{attribute 'reflection'}
FUNCTION_BLOCK ABSTRACT Objective
VAR_INPUT

	Mediator					: REFERENCE TO Mediator;	

END_VAR
VAR

    internalRegisteredMoverCount 	: USINT;
   
    internalRegisteredMovers 		: ARRAY[1..Param.NUM_MOVERS] OF POINTER TO Mover;

	{attribute 'hide'}
    ErrorMover 					: ErrorMover;
	
    {attribute 'instance-path'}
    {attribute 'noinit'}
    InstancePath 				: STRING; // Unique variable path of the instance	
END_VAR
VAR_OUTPUT
END_VAR

PROPERTY CurrentMover : Reference to Mover
GET

// If no real mover can be returned as Current, return an imposter instead to output error messages
IF __ISVALIDREF( CurrentMover ) = FALSE THEN
	ErrorMover.SourceInstancePath	:= THIS^.InstancePath;
	CurrentMover					REF= ErrorMover;
END_IF
END_GET
END_PROPERTY

{attribute 'monitoring' := 'call'}
PROPERTY RegisteredMoverCount : USINT
GET
VAR
    i : INT;
END_VAR
RegisteredMoverCount := 0;

FOR i := 1 to Param.NUM_MOVERS DO

    IF internalRegisteredMovers[i] <> 0 THEN
        RegisteredMoverCount := RegisteredMoverCount + 1;
    END_IF

END_FOR
END_GET
END_PROPERTY

PROPERTY RegisteredMovers : ARRAY[0..Param.NUM_MOVERS - 1] OF POINTER TO Mover
GET
RegisteredMovers := internalRegisteredMovers;
END_GET
END_PROPERTY

METHOD RegisterMover : BOOL
VAR_INPUT
    NewMover : REFERENCE TO Mover;
END_VAR

VAR
    i              : ULINT;
    duplicateFound : BOOL;
    emptyIDX       : ulint;
END_VAR
(*
	Add a mover to a list of movers tracked by the objective.
	Movers can't be added multiple times, so check for duplicates
	Movers can't overwrite others in the list, so check that the array element is clear
*)

IF __ISVALIDREF(NewMover) THEN // validate reference

    duplicateFound            := FALSE; // default to false, counterexample below
    internalRegisteredMoverCount := 0;     // reset to zero, incremented below

    FOR i := 1 TO SIZEOF(internalRegisteredMovers) / SIZEOF(internalRegisteredMovers[i]) DO
        IF internalRegisteredMovers[i] <> 0 THEN
            IF ADR(NewMover) = internalRegisteredMovers[i] THEN
                duplicateFound := TRUE; // this mover already tracked
            END_IF

            internalRegisteredMoverCount := internalRegisteredMoverCount + 1;
        ELSE
			// track the first empty index
			IF (emptyIDX = 0) THEN
				emptyIDX	:= i;
			END_IF;
        END_IF
    END_FOR

    IF duplicateFound = FALSE THEN
        internalRegisteredMovers[emptyIDX] := ADR(NewMover); // new mover goes into open array element
        internalRegisteredMoverCount       := internalRegisteredMoverCount + 1;
    END_IF

ELSE
    ADSLOGSTR(ADSLOG_MSGTYPE_LOG, 'Error: Mover registration input is invalid', '');
END_IF
END_METHOD

METHOD RegisterMoverList : BOOL
VAR_INPUT
    NewMoverList : iMoverList;
END_VAR
VAR
    i                : ULINT;
    duplicateFound   : BOOL;
    emptyIDX         : USINT;
    arrRegisteredMovers : ARRAY[0..Param.NUM_MOVERS - 1] OF POINTER TO Mover;
END_VAR
(*
	Adds an entire MoverList to the Tracked Movers of the objective.
*)

arrRegisteredMovers := NewMoverList.RegisteredMovers;

// IF __ISVALIDREF( NewMoverList ) THEN
IF NewMoverList <> 0 THEN
    FOR i := 1 TO SIZEOF(arrRegisteredMovers) / SIZEOF(arrRegisteredMovers[0]) DO

        THIS^.RegisterMover(arrRegisteredMovers[i]^);

    END_FOR
END_IF
END_METHOD

METHOD UnregisterAll : BOOL
VAR_INPUT
END_VAR
VAR
    i : USINT;
END_VAR
// Blow out the tracked mover array
memset(ADR(internalRegisteredMovers), 0, SIZEOF(internalRegisteredMovers));
END_METHOD

METHOD UnregisterCurrent : BOOL
VAR_INPUT
END_VAR
THIS^.UnregisterMover(CurrentMover);
END_METHOD

METHOD UnregisterMover : BOOL
VAR_INPUT
    RemovingMover : REFERENCE TO Mover;
END_VAR
VAR
    i              : dint;
END_VAR
(*
	Remove a mover to a list of movers tracked by the objective.
	Only movers in the list can be removed, otherwise nothing happens
*)

//	IF RemovingMover <> 0 THEN			// validate pointer
IF __ISVALIDREF(RemovingMover) THEN

    internalRegisteredMoverCount := 0;

    FOR i := 1 TO SIZEOF(internalRegisteredMovers) / SIZEOF(internalRegisteredMovers[1]) DO
        IF internalRegisteredMovers[i] <> 0 THEN // validate pointer

            internalRegisteredMoverCount := internalRegisteredMoverCount + 1;

            IF ADR(RemovingMover) = internalRegisteredMovers[i] THEN
                internalRegisteredMovers[i]  := 0; // remove the pointer
                internalRegisteredMoverCount := internalRegisteredMoverCount - 1;
            END_IF

        END_IF
    END_FOR

ELSE
    ADSLOGSTR(ADSLOG_MSGTYPE_LOG, 'Error: Mover input is invalid', '');
END_IF
END_METHOD

END_FUNCTION_BLOCK

(* stored: Version 1.1.0.1, ProductVersion 3.1.4026.8
   POU Objective: Id {72371872-54aa-4f25-a82d-ba585015a7c5}, SpecialFunc None
   Folder Methods: Id {4ed72c29-121a-4b01-8ee9-80f4e3e37fcf}
   Folder Properties: Id {a322a947-e1f7-42e0-b1f3-cb1cbcbf3e25}
   Property CurrentMover: Id {99a54d83-41c7-49ce-a206-e4c6b3a981c8}
   Get Get: Id {8bd4cff1-d1fd-42f7-b813-8805845e8ad0}
   Property RegisteredMoverCount: Id {610e1915-c97a-4bca-998c-120d922f3eee}
   Get Get: Id {7832ece5-c334-41ff-a04f-4af0717e7184}
   Property RegisteredMovers: Id {f2e27676-d8a8-4b3f-968b-790753e7621e}
   Get Get: Id {2692defb-0744-4a89-a02c-657d915f8a30}
   Method RegisterMover: Id {8354cf16-6187-4fe4-976a-42e2fe3b8399}
   Method RegisterMoverList: Id {97f69758-a5f2-4092-9f2f-11848d10cf56}
   Method UnregisterAll: Id {8fb61f33-6bbe-4b93-92b5-f08c59b94375}
   Method UnregisterCurrent: Id {f5252866-1ebe-4ec3-aeab-827236ab79ab}
   Method UnregisterMover: Id {18c8f6fd-1567-45b0-85d6-dc2464792b83} *)
